Universal Robots PolyScope program: 25-script_file.urp

ProgramRoot directory=/home/ur/ursim-3.1/programs/25-script_file; kinematics=(a=[0, -0.425, -0.39225, 0, 0, 0], d=[0.08916, 0, 0, 0.10915, 0.09465, 0.0823], alpha=[1.5708, 0, 0, 1.5708, -1.5708, 0], deltaTheta=[0, 0, 0, 0, 0, 0], status=notInitialized); lastSavedInVersion=(project__name=Polyscope, major__version=3, minor__version=1, svn__revision=17195, build__date=Mar 11 2015, 13:02:28); name=25-script_file; programVersion=(project__name=Polyscope, major__version=3, minor__version=1, svn__revision=17195, build__date=Mar 11 2015, 13:02:28); robotEnvironmentFileName=default; serialNumberRobot=2014350001
  MainProgram cartesianAcceleration=1.2; cartesianSpeed=0.25; jointAcceleration=1.3962634015954636; jointSpeed=1.0471975511965976; sharedProcessMoveBlendRadius=0.025; motionType=JOINT_SPACE
    Script type=1; cachedFileContents=movej([-1.6007002035332292, -1.5827531569708118, -2.093159502954533, -1.0621873442540695, 1.5951000452051884, -0.030999962444354878], a=1.3962634015954636, v=1.0471975511965976)
      |     movej([-1.6007002035724085, -1.7271001974688929, -2.2029998938189905, -0.8079999128924769, 1.5951000452041626, -0.03099996248354131], a=1.3962634015954636, v=1.0471975511965976); scriptFile=/home/ur/ursim-3.1/programs/25-script_file/test.script
